{attribute 'linkalways'} 
{attribute 'no_explicit_call' := 'This FB is a CLASS and must be accessed using methods or properties'}
{attribute 'enable_dynamic_creation'}
FUNCTION_BLOCK FINAL ADD_REAL EXTENDS Node
VAR
	in1 : _REAL(0.0);
	in2 : _REAL(0.0);
	out : _REAL(0.0);
END_VAR

METHOD PUBLIC Clone : I_Node
VAR
	pNode : POINTER TO ADD_REAL;
END_VAR
pNode := __NEW(ADD_REAL);
Clone := pNode^;
END_METHOD

METHOD FB_init : BOOL
VAR_INPUT
	bInitRetains : BOOL; // if TRUE, the retain variables are initialized (warm start / cold start)
	bInCopyCode : BOOL;  // if TRUE, the instance afterwards gets moved into the copy code (online change)
END_VAR
AddInput('in1',THIS^.in1);
AddInput('in2',THIS^.in2);
AddOutput('out', THIS^.out);
END_METHOD

METHOD PROTECTED OnExecute
VAR
END_VAR
out.Value := in1.Value + in2.Value;
END_METHOD

END_FUNCTION_BLOCK

(* stored: Version 1.1.0.1, ProductVersion 3.1.4024.15
   POU ADD_REAL: Id {dfcb69dc-5852-44f4-936f-d93c5c186a48}, SpecialFunc None
   Folder Constructor: Id {e434c91d-47e2-443c-b3a3-fb6e1a825fe4}
   Method Clone: Id {84a736a4-78f6-4f91-8dc1-e0f12daf5cd6}
   Method FB_init: Id {d33e6903-ac91-43cf-8962-a5a4c1e19fe1}
   Method OnExecute: Id {3080a5cc-ed48-445a-8486-ba3c128e3ef5} *)
